{attribute 'GeneratedUsingTerminal: EK1122-0000-0018'}
{attribute addProperty BoxType "EK1122-0000-0018"}
{attribute addProperty Id "Beckhoff_EK13xxsub_EK1100EK1100_AB5A94672A_0001_EK1300_0000_0017EK1300_0DA715C26"}
{attribute addProperty CRC "506920058"}
{attribute addProperty Size "8"}
TYPE Beckhoff_EK13xxEK1122_1E36FC7A EXTENDS EK1122_AB5A9467 :
STRUCT
	{attribute addProperty Name "Beckhoff_EK13xxsub_EK1100"}
	{attribute addProperty PreviousPort "Beckhoff EK13xxEK1122 : D"}
	Beckhoff_EK13xxsub_EK1100 : EK1100_AB5A9467;
	{attribute addProperty Name "A_0001_EK1300_0000_0017"}
	{attribute addProperty PreviousPort "Beckhoff EK13xxsub EK1100 : C"}
	A_0001_EK1300_0000_0017 : EK1300_0DA715C2;
END_STRUCT
END_TYPE

(* stored: Version 1.2.0.0, ProductVersion 3.1.4024.9
   DUT Beckhoff_EK13xxEK1122_1E36FC7A: Id {e2ed047a-78b1-4045-a292-ad3e03d6868b} *)
